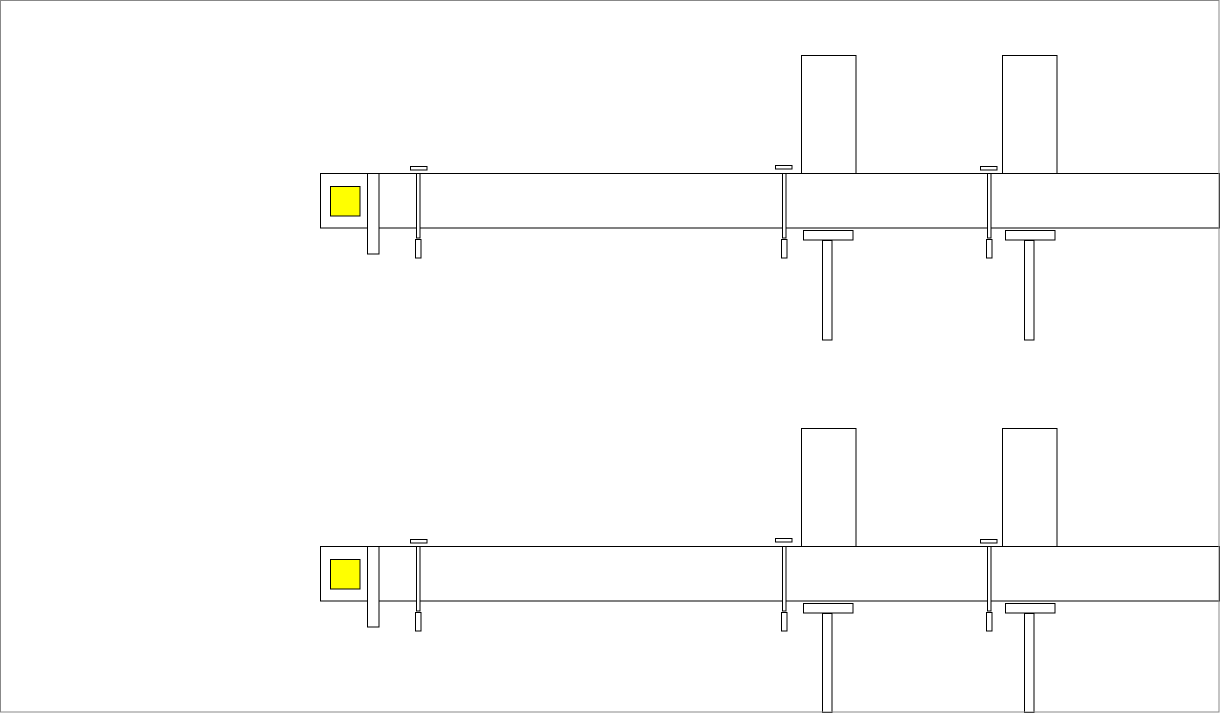
VISUALIZATION Visualization  // 1220x713
    Rectangle (801,55 55x120)
    Rectangle (1002,55 55x120)
    Rectangle (320,173 900x55)
    Rectangle (330,186 30x30), colour toggle: MAIN.Mashine1Boxes[4].IsMetal
        p3560616238: MAIN.Mashine1Boxes[4].PositionHOZ
        p2738717112: MAIN.Mashine1Boxes[4].PositionVTK
    Rectangle (330,186 30x30), colour toggle: MAIN.Mashine1Boxes[3].IsMetal
        p3560616238: MAIN.Mashine1Boxes[3].PositionHOZ
        p2738717112: MAIN.Mashine1Boxes[3].PositionVTK
    Group (803,230 50x110)
        p2738717112: MAIN.MyMashine1.FirstAxes.AxesPosition
        Rectangle (0,0 50x10)
        Rectangle (19,10 10x100)
    Group (1005,230 50x110)
        p2738717112: MAIN.MyMashine1.SecondAxes.AxesPosition
        Rectangle (0,0 50x10)
        Rectangle (19,10 10x100)
    Rectangle (330,186 30x30), colour toggle: MAIN.Mashine1Boxes[2].IsMetal
        p3560616238: MAIN.Mashine1Boxes[2].PositionHOZ
        p2738717112: MAIN.Mashine1Boxes[2].PositionVTK
    Rectangle (416,173 4x65)
    Rectangle (782,173 4x65)
    Rectangle (987,173 4x65)
    Rectangle (367,173 12x81)
        p2738717112: MAIN.MyMashine1.MyGate.GatePosition
    Rectangle (410,166 17x4)
    Rectangle (775,165 17x4)
    Rectangle (980,166 17x4)
    Rectangle (415,239 6x19)
    Rectangle (781,239 6x19)
    Rectangle (986,239 6x19)
    Rectangle (330,186 30x30), colour toggle: MAIN.Mashine1Boxes[1].IsMetal
        p3560616238: MAIN.Mashine1Boxes[1].PositionHOZ
        p2738717112: MAIN.Mashine1Boxes[1].PositionVTK
    Rectangle (801,428 55x120)
    Rectangle (1002,428 55x120)
    Rectangle (320,546 900x55)
    Rectangle (330,559 30x30), colour toggle: MAIN.Mashine2Boxes[4].IsMetal
        p3560616238: MAIN.Mashine2Boxes[4].PositionHOZ
        p2738717112: MAIN.Mashine2Boxes[4].PositionVTK
    Rectangle (330,559 30x30), colour toggle: MAIN.Mashine2Boxes[3].IsMetal
        p3560616238: MAIN.Mashine2Boxes[3].PositionHOZ
        p2738717112: MAIN.Mashine2Boxes[3].PositionVTK
    Group (803,603 50x110)
        p2738717112: MAIN.MyMashine2.FirstAxes.AxesPosition
        Rectangle (0,0 50x10)
        Rectangle (19,10 10x100)
    Group (1005,603 50x110)
        p2738717112: MAIN.MyMashine2.SecondAxes.AxesPosition
        Rectangle (0,0 50x10)
        Rectangle (19,10 10x100)
    Rectangle (330,559 30x30), colour toggle: MAIN.Mashine2Boxes[2].IsMetal
        p3560616238: MAIN.Mashine2Boxes[2].PositionHOZ
        p2738717112: MAIN.Mashine2Boxes[2].PositionVTK
    Rectangle (416,546 4x65)
    Rectangle (782,546 4x65)
    Rectangle (987,546 4x65)
    Rectangle (367,546 12x81)
        p2738717112: MAIN.MyMashine2.MyGate.GatePosition
    Rectangle (410,539 17x4)
    Rectangle (775,538 17x4)
    Rectangle (980,539 17x4)
    Rectangle (415,612 6x19)
    Rectangle (781,612 6x19)
    Rectangle (986,612 6x19)
    Rectangle (330,559 30x30), colour toggle: MAIN.Mashine2Boxes[1].IsMetal
        p3560616238: MAIN.Mashine2Boxes[1].PositionHOZ
        p2738717112: MAIN.Mashine2Boxes[1].PositionVTK
END_VISUALIZATION

(* stored: Version 1.1.0.1, ProductVersion 3.1.4024.3
   Visu Visualization: Id {1553f28f-69ae-469d-ad25-680a38e0067c} *)
